FUNCTION_BLOCK FieldsToServiceQueryForm (* Translate individual fields to a Service Query Form type *)
  (* Standard: 61499-2; Description: Copyright (c) 2018 fortiss GmbH This program and the accompanying materials are made available under the terms of the Eclipse Public License 2.0 which is available at https://www.eclipse.org/legal/epl-2.0/ SPDX-License-Identifier: EPL-2.0 *)
  (* Version 1.0, 2018-09-21, Jose Cabral, fortiss GmbH *)
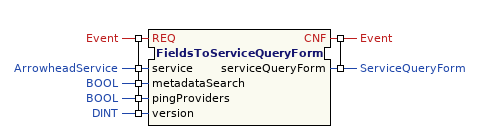
  EVENT_INPUT
    REQ WITH service, version, pingProviders, metadataSearch; (* Create Service Query Form *)
  END_EVENT
  EVENT_OUTPUT
    CNF WITH serviceQueryForm; (* Service Query Form created *)
  END_EVENT
  VAR_INPUT
    service : ArrowheadService; (* The Arrowhead Service object that is looked for (SD and supported IDD-s) *)
    metadataSearch : BOOL; (* True, if service metadata shall be taken into account during query *)
    pingProviders : BOOL; (* True, if the selected (query fitting) Application Systems shall be pinged to see if they’re alive *)
    version : DINT; (* The minimum version of the Service we are looking for *)
  END_VAR
  VAR_OUTPUT
    serviceQueryForm : ServiceQueryForm; (* Created Service Query Form *)
  END_VAR
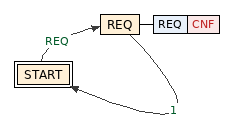
  EC_STATES
    START; (* Initial State *)
    REQ : REQ -> CNF; (* Initialization *)
  END_STATES
  EC_TRANSITIONS
    START TO REQ := REQ;
    REQ TO START := 1;
  END_TRANSITIONS
  ALGORITHM REQ IN ST: (* Initialization algorithm *)
serviceQueryForm.service := service;
serviceQueryForm.metadataSearch := metadataSearch;
serviceQueryForm.pingProviders := pingProviders;
serviceQueryForm.version := version;
  END_ALGORITHM
END_FUNCTION_BLOCK
